{attribute 'GeneratedUsingTerminal: EP2001-1000-0016'}
{attribute addProperty BoxType "EP2001-1000-0016"}
{attribute addProperty Id "EtcSlaveTerminalBaseGroup_0AT %Q*Group_99EF3D304Group_1AT %Q*Group_8FCDB3954WcStateAT %I*WcState_0B2B16F91InfoDataAT %I*InfoData_6F19DB2B2"}
{attribute addProperty CRC "3945159138"}
{attribute addProperty Size "11"}
TYPE EP2001_EB2659E2 EXTENDS EtcSlaveTerminalBase :
STRUCT
	{attribute addProperty Name "Group_0"}
	Group_0 : Group_99EF3D30;
	{attribute addProperty Name "Group_1"}
	Group_1 : Group_8FCDB395;
	{attribute addProperty Name "WcState"}
	WcState : WcState_0B2B16F9;
	{attribute addProperty Name "InfoData"}
	InfoData : InfoData_6F19DB2B;
END_STRUCT
END_TYPE

(* stored: Version 1.2.0.0, ProductVersion 3.1.4024.9
   DUT EP2001_EB2659E2: Id {95a449b0-12d2-4049-a285-76db6bbfd6d6} *)
